{attribute 'OPC.UA.DA.StructuredType' := '1'}
TYPE ST_UnderfloorHeatingSetParameters :
STRUCT
	bHeatingModeAlgorithm : BOOL;
	bHeatingModeManual : BOOL;
END_STRUCT
END_TYPE

(* stored: Version 1.1.0.1, ProductVersion 3.1.4024.10
   DUT ST_UnderfloorHeatingSetParameters: Id {af258353-03b2-46dd-afd7-9b0deec3f899} *)
